// TIA Portal V19 export
DATA_BLOCK "MODE SELECTION DB"   // DB3
{ S7_Optimized_Access := 'TRUE' }
// stored: MemoryReserve 100
   VAR
      STANDBY : Bool;
      AUTO : Bool;
      MANUAL : Bool;
      START : Bool;
      STOP : Bool;
   END_VAR
   VAR RETAIN
      "MODE BUFF" : Int;
      "PROCESS BUFF" : Int;
   END_VAR
BEGIN
END_DATA_BLOCK
